// TwinCAT 3 PLC project TcoInspectors
// Title: TcoInspectors
// Company: Vortex.Library
// ProjectVersion: 0.6.0.913
// ProgramVersion: 3.1.4023.0
// libraries:
//   Tc2_Standard, * (Beckhoff Automation GmbH)
//   Tc2_System, * (Beckhoff Automation GmbH)
//   Tc2_Utilities, * (Beckhoff Automation GmbH)
//   Tc3_Module, * (Beckhoff Automation GmbH)
//   TcoCore, 0.6.0.913 (Vortex.Library)
// project tree:
//   / PlcTask.TcTTO
//   POUs/TcoInspector/ eTcoInspectorFailMode.TcDUT, IInspector.TcIO, IOnFail.TcIO, TcoComprehensiveResult.TcDUT, TcoInspector.TcPOU, TcoInspectorDialog.TcPOU, TcoInspectorTask.TcPOU, TcoInspectorData.TcDUT
//   POUs/TcoAnalogueInspector/ ITcoAnalogueInspector.TcIO, TcoAnalogueInspectorData.TcDUT, TcoAnalogueInspector.TcPOU
//   POUs/TcoDataInspector/ ITcoDataInspector.TcIO, TcoDataInspectorData.TcDUT, TcoDataInspector.TcPOU
//   POUs/ eOverallResult.TcDUT, eInspectorResult.TcDUT, MAIN.TcPOU
//   POUs/TcoDigitalInspector/ ITcoDigitalInspector.TcIO, TcoDigitalInspector.TcPOU, TcoDigitalInspectorData.TcDUT
//   POUs/TcoInspectionGroup/ ITcoInspectionGroup.TcIO, ITcoInspectionGroupAct.TcIO, TcoInspectionGroup.TcPOU
// real-time tasks:
//   TASK PlcTask: cycle T#10ms, priority 20, ADS port 350
//   TASK PlcTask1: cycle T#10ms, priority 21, ADS port 351

CONFIGURATION TcoInspectors
    RESOURCE PLC ON TwinCAT3
        TASK PlcTask(INTERVAL := T#10ms, PRIORITY := 20);
        PROGRAM MAIN WITH PlcTask : MAIN;
    END_RESOURCE
END_CONFIGURATION

// ---- POUs/TcoInspector/eTcoInspectorFailMode.TcDUT
{attribute 'qualified_only'}
{attribute 'strict'}
TYPE
    eTcoInspectorFailMode :
    (
        // On failed continues in the sequence but data are set to failed.
        CarryOn := 0,
        // Jump to specific step after first fail.
        JumpTo := 10,
        // Restores origin after first fail.
        Terminate := 20,
        // Retry when failed given number of times and continues in the sequence. Data are set to failed.
        RetryThenCarryOn := 30,
        // Retry, when failed given number of times abort sequence and continue in specifed step. Data are set to failed.
        RetryThenJumpTo := 40,
        // Retry, when failed given number of times abort sequence and continue with restore section. Data are set to failed.
        RetryThenTeminate := 50

    );
END_TYPE

// ---- POUs/TcoInspector/TcoComprehensiveResult.TcDUT
TYPE TcoComprehensiveResult :
STRUCT
    Result : eOverallResult;
    Failures : STRING(255);
    ErrorCodes : STRING(255);
END_STRUCT
END_TYPE

// ---- POUs/TcoInspector/TcoInspectorData.TcDUT
(*~
    <docu>
        <summary>
            Defines data commonly used accross different types of inspectors.
        </summary>
    </docu>
~*)
{attribute 'qlik_entity:Checks'}
{attribute 'qlik_ref_value_field:CheckName = AttributeHumanReadable'}
{attribute 'qlik_ref_value_field:StationName = AttributeQlikGroup'}
TYPE TcoInspectorData :
STRUCT
    (*~
        <docu>
        <summary>
            Inspection timestamp.
        </summary>
        </docu>
    ~*)
    {attribute addProperty Name "<#Time stamp#>"}
    {attribute clr [RenderIgnore("Control", "ShadowControl")]}
    {attribute 'qlik_load:TimeStamp'}
    TimeStamp : DT;
    (*~
        <docu>
        <summary>
            Pass time, elapses when the measured value has required value (see `ReuiredStatus`).
            The signal must have required value continuosly for this time span for the check to pass.
        </summary>
        </docu>
    ~*)
    {attribute addProperty Name "<#Stab.Time#>"}
    {attribute addProperty ToolTip "<#Stabilisation time. The inspection will pass when the condition is met continuously for the duration of this timespan.#>"}
    {attribute 'qlik_load:PassedTime'}
    PassTime : TIME;
    (*~
        <docu>
        <summary>
            Fail time. Is the maximum test duration (or timeout). If the condition for the successul test is not met within this time, the test fails.
        </summary>
        </docu>
    ~*)
    {attribute addProperty Name "<#Timeout#>"}
    {attribute addProperty ToolTip "<#Timeout. Maximal duration of the inspection within which the condition must be met.#>"}
    {attribute 'qlik_load:FailedTime'}
    FailTime : TIME;
    (*~
        <docu>
        <summary>
            Test result.
        </summary>
        </docu>
    ~*)
    {attribute addProperty Name "<#Result#>"}
    {attribute clr [RenderIgnore("Control", "ShadowControl")]}
    {attribute addProperty ToolTip "<#Result of the inspection.#>"}
    {attribute 'qlik_load:Result'}
    Result : eInspectorResult;
    (*~
        <docu>
        <summary>
            Test is excluded from evaluation. If TRUE the check is excluded, the test will run and provide detected value.
            Evaluation of excluded test should be handled by user code.
        </summary>
        </docu>
    ~*)
    {attribute addProperty Name "<#Exclude#>"}
    {attribute addProperty ToolTip "<#Inspection is excluded from the evaluation. The test will however run and provide detected value.#>"}
    {attribute 'qlik_load:IsExcluded'}
    IsExcluded : BOOL;
    (*~
        <docu>
        <summary>
            Test is bypassed, no eveluation occurs.
            Evaluation of excluded test should be handled by user code.
        </summary>
        </docu>
    ~*)
    {attribute addProperty Name "<#Bypass#>"}
    {attribute addProperty ToolTip "<#Test is bypassed, no eveluation occurs.#>"}
    {attribute 'qlik_load:IsByPassed'}
    IsByPassed : BOOL;
    (*~
        <docu>
        <summary>
            Verbatim description of the failure.
        </summary>
        </docu>
    ~*)
    {attribute addProperty Name "<#Failure description#>"}
    {attribute addProperty ToolTip "<#Brief failure desciption#>"}
    {attribute 'qlik_ignore'}
    FailureDescription : STRING(100);
    (*~
        <docu>
        <summary>
            Counter of allowed inspections.
        </summary>
        </docu>
    ~*)
    {attribute addProperty Name "<#Re-tries#>"}
    {attribute addProperty ToolTip "<#Inspection will repeat given number of times when inspection fails.#>"}
    {attribute 'qlik_load:NumberOfAllowedRetries'}
    NumberOfAllowedRetries : UINT;
    (*~
        <docu>
        <summary>
            Counter inspections.
        </summary>
        </docu>
    ~*)
    {attribute addProperty Name "<#Attempts#>"}
    {attribute addProperty ToolTip "<#Re-tries counter, count the number of times the inspection run on this inspector instance.#>"}
    {attribute 'qlik_load:RetryAttemptsCount'}
    RetryAttemptsCount : UINT;
    (*~
        <docu>
        <summary>
            Error code.
        </summary>
        </docu>
    ~*)
    {attribute addProperty Name "<#Code#>"}
    {attribute addProperty ToolTip "<#Arbitrary error code for this inspection#>"}
    {attribute 'qlik_load:ErrorCode'}
    ErrorCode : STRING(20);
END_STRUCT
END_TYPE

// ---- POUs/TcoDataInspector/TcoDataInspectorData.TcDUT
{attribute addProperty Name "AnalogueCheckerData"}
{attribute 'qlik_entity:Checks'}
{attribute 'qlik_ref_value_field:CheckName = AttributeHumanReadable'}
{attribute 'qlik_ref_value_field:StationName = AttributeQlikGroup'}
{attribute 'qlik_value_field:CheckType = Analogue'}
TYPE TcoDataInspectorData EXTENDS TcoInspectorData :
STRUCT
    (*~
        <docu>
        <summary>
            Required status for the check to Pass.
        </summary>
        </docu>
        ~*)
    {attribute addProperty Name "<#Required#>"}
    {attribute addProperty ToolTip "<#Required status for inspection to pass. Can contain pattern string when `Star notation is enabled`#>"}
    {attribute 'qlik_load:RequiredStatus'}
    RequiredStatus : STRING(255);
    (*~
        <docu>
        <summary>
            Detected status.
        </summary>
        </docu>
        ~*)
    {attribute addProperty  Name "<#Detected#>"}
    {attribute addProperty ToolTip "<#Detected data#>"}
    {attribute clr [RenderIgnore("Control", "ShadowControl", "ControlSlim", "ShadowControlSlim")]}
    {attribute 'qlik_load:Measured'}
    DetectedStatus : STRING(255);
    (*~
        <docu>
        <summary>
            When enabled (`true`) the date are evaluating with simple pattern matching.
        </summary>
        </docu>
        ~*)
    {attribute addProperty  Name "<*>"}
    {attribute addProperty ToolTip "<#Required status for inspection to pass. Can contain pattern string when `Star notation is enabled`#>"}
    {attribute 'qlik_load:Measured'}
    StarNotationEnabled : BOOL;
END_STRUCT
END_TYPE

// ---- POUs/eOverallResult.TcDUT
{attribute 'qualified_only'}
{attribute 'strict'}
TYPE eOverallResult :
(
    NoAction := 0,
    InProgress := 10,
    Passed := 20,
    Failed := 30
);
END_TYPE

// ---- POUs/TcoAnalogueInspector/TcoAnalogueInspectorData.TcDUT
{attribute addProperty Name "AnalogueCheckerData"}
{attribute addProperty Units ""}
{attribute 'qlik_entity:Checks'}
{attribute 'qlik_ref_value_field:CheckName = AttributeHumanReadable'}
{attribute 'qlik_ref_value_field:StationName = AttributeQlikGroup'}
{attribute 'qlik_value_field:CheckType = Analogue'}
TYPE TcoAnalogueInspectorData EXTENDS TcoInspectorData :
STRUCT
    (*~
        <docu>
        <summary>
            Required minimum value for the inspection to pass.
        </summary>
        </docu>
        ~*)
    {attribute addProperty  Name "<#Min.#>"}
    {attribute 'qlik_load:Minimum'}
    {attribute addProperty ToolTip "<#Min. value for the inspection to pass.#>"}
    RequiredMin : LREAL;
    (*~
        <docu>
        <summary>
            Detected status.
        </summary>
        </docu>
        ~*)
    {attribute addProperty  Name "<#Detected#>"}
    {attribute clr [RenderIgnore("Control", "ShadowControl", "ControlSlim", "ShadowControlSlim")]}
    {attribute addProperty ToolTip "<#Detected value#>"}
    {attribute 'qlik_load:Measured'}
    DetectedStatus : LREAL;
    (*~
        <docu>
        <summary>
            Required maximum value for the inspection to pass.
        </summary>
        </docu>
        ~*)
    {attribute addProperty  Name "<#Max.#>"}
    {attribute 'qlik_load:Maximum'}
    {attribute addProperty ToolTip "<#Max. value for the inspection to pass.#>"}
    RequiredMax : LREAL;
END_STRUCT
END_TYPE

// ---- POUs/TcoDigitalInspector/TcoDigitalInspectorData.TcDUT
{attribute addProperty Name "LogicCheckerData"}
{attribute 'qlik_value_field:CheckType = Logic'}
TYPE TcoDigitalInspectorData EXTENDS TcoInspectorData :
STRUCT
    (*~
        <docu>
        <summary>
            Required status for the check to Pass.
        </summary>
        </docu>
        ~*)
    {attribute addProperty Name "<#Required#>"}
    {attribute addProperty ToolTip "<#Sets the required status for the inspection to pass.#>"}
    {attribute 'qlik_load:RequiredStatus'}
    RequiredStatus : BOOL;
    (*~
        <docu>
        <summary>
            Detected status.
        </summary>
        </docu>
    ~*)
    {attribute addProperty Name "<#Detected#>"}
    {attribute clr [RenderIgnore("Control", "ShadowControl", "ControlSlim", "ShadowControlSlim")]}
    {attribute addProperty ToolTip "<#Displays detected status of this check.#>"}
    {attribute 'qlik_load:DetectedStatus'}
    DetectedStatus : BOOL;
END_STRUCT
END_TYPE

// ---- POUs/eInspectorResult.TcDUT
{attribute 'qualified_only'}
{attribute 'strict'}
TYPE eInspectorResult :
(
    NoAction := 0,
    Running := 10,
    Passed := 20,
    Failed := 30,
    Inconclusive := 35,
    Excluded := 40,
    Bypassed := 50
);
END_TYPE

// ---- POUs/TcoInspector/IInspector.TcIO
INTERFACE IInspector EXTENDS __SYSTEM.IQueryInterface

PROPERTY Busy : BOOL
GET
END_GET
END_PROPERTY

(*~
	<docu>
		<summary>
			Gets common data settings of inspectors.
		</summary>			
	</docu>	
~*)
PROPERTY CommonData : REFERENCE TO TcoInspectorData
GET
END_GET
END_PROPERTY

PROPERTY Coordinator : TcoCore.ITcoCoordinator
GET
END_GET
END_PROPERTY

PROPERTY Done : BOOL
GET
END_GET
END_PROPERTY

METHOD HideOverride : IInspector
END_METHOD

METHOD HideRetry : IInspector
END_METHOD

METHOD HideTerminate : IInspector
END_METHOD

PROPERTY Identity : ULINT
GET
END_GET
END_PROPERTY

METHOD Instruct : IInspector
VAR_INPUT
	inInstruction:STRING(255);
END_VAR
END_METHOD

METHOD InstructWithImage : IInspector
VAR_INPUT
	inImageSource:STRING(255);
	inHeight:REAL;
	inWidth:REAL;
END_VAR
END_METHOD

METHOD OnFail : IOnFail
END_METHOD

PROPERTY OverInspected : BOOL
GET
END_GET
END_PROPERTY

PROPERTY Result : eInspectorResult
GET
END_GET
END_PROPERTY

(*~
	<docu>
		<summary>
			Updates comprehensive result. The comprehensive result is set to `Failed` when any inspection fails or is inconclusive.
			Any bypassed or excluded inspection are not taken in the account.			
		</summary>			
	</docu>	
~*)
METHOD UpdateComprehensiveResult : IInspector
VAR_IN_OUT
	(*~
	<docu>
		<summary>
			Comprehensive result data structure to be updated.	
		</summary>			
	</docu>	
	~*)
    inoResult : TcoComprehensiveResult;
END_VAR
END_METHOD

(*~
	<docu>
		<summary>
			Provide information about the Inspector name (if there are multiple inspectors, only the failed ones will be displayed).  (e.g. {attribute addProperty Name "Bolt presence inspection"})
		</summary>			
	</docu>	
~*)
METHOD WithDescription : IInspector
END_METHOD

(*~
	<docu>
		<summary>
			Provide information about ErrorCode (if there are multiple inspectors, only the failed ones will be displayed). Error codes shoud be defined in Inspectors
		</summary>			
	</docu>	
~*)
METHOD WithErrorCode : IInspector
END_METHOD

(*~
	<docu>
		<summary>
			Provide information about Failure Description (if there are multiple inspectors, only the failed ones will be displayed). Failure description shoud be defined in Inspectors.
		</summary>			
	</docu>	
~*)
METHOD WithFailureDescription : IInspector
END_METHOD

END_INTERFACE

// ---- POUs/TcoInspector/IOnFail.TcIO
INTERFACE IOnFail EXTENDS __SYSTEM.IQueryInterface

METHOD CarryOn : BOOL
END_METHOD

METHOD Dialog : BOOL
VAR_INPUT
	inRetryStep : INT;
END_VAR
END_METHOD

METHOD DialogWithExternalClose : BOOL
VAR_INPUT
	inRetryStep : INT;
	inRetrySignal:BOOL;
	inTerminateSignal : BOOL;
END_VAR
END_METHOD

METHOD Evaluate : BOOL
VAR_INPUT
	inFromState : INT;
	inFailMode : eTcoInspectorFailMode;
    inToState : INT;
END_VAR
END_METHOD

METHOD Retry : BOOL
VAR_INPUT
	inFromState : INT;
END_VAR
END_METHOD

METHOD RetryThenTerminate : BOOL
VAR_INPUT
	inFromState : INT;
END_VAR
END_METHOD

METHOD Terminate : BOOL
END_METHOD

END_INTERFACE

// ---- POUs/TcoAnalogueInspector/ITcoAnalogueInspector.TcIO
INTERFACE ITcoAnalogueInspector

(*~
<docu>
<summary>
	Inspects the signal and evaluates that it matches the value set in `RequiredStatus`.
</summary>
<returns>
	Returns the interface with information about the state of inspection.
</returns>
</docu>
~*)
METHOD Inspect : IInspector
VAR_INPUT
    Status : LREAL;
END_VAR
END_METHOD

END_INTERFACE

// ---- POUs/TcoDataInspector/ITcoDataInspector.TcIO
INTERFACE ITcoDataInspector

(*~
<docu>
<summary>
	Inspects the signal and evaluates that it matches the value set in `RequiredStatus`.
</summary>
<returns>
	Returns the interface with information about the state of inspection.
</returns>
</docu>
~*)
METHOD Inspect : IInspector
VAR_INPUT
    Status : STRING(255);
END_VAR
END_METHOD

END_INTERFACE

// ---- POUs/TcoDigitalInspector/ITcoDigitalInspector.TcIO
INTERFACE ITcoDigitalInspector

(*~
<docu>
<summary>
	Inspects the signal and evaluates that it matches the value set in `RequiredStatus`.
</summary>
<returns>
	Returns the interface with information about the state of inspection.
</returns>
</docu>
~*)
METHOD Inspect : IInspector
VAR_INPUT
    Status : BOOL;
END_VAR
END_METHOD

END_INTERFACE

// ---- POUs/TcoInspectionGroup/ITcoInspectionGroup.TcIO
INTERFACE ITcoInspectionGroup

PROPERTY Done : BOOL
GET
END_GET
END_PROPERTY

METHOD Inspect : ITcoInspectionGroup
VAR_INPUT
    Inspector : IInspector;
END_VAR
END_METHOD

METHOD NormalizeRetries : ITcoInspectionGroup
VAR_INPUT
	inoInspection : IInspector;
END_VAR
END_METHOD

METHOD OnFail : IOnFail
END_METHOD

(*~
	<docu>
		<summary>
			Updates comprehensive result. The comprehensive result is set to `Failed` when any inspection fails or is inconclusive.
			Any bypassed or excluded inspection are not taken in the account.
		</summary>
	</docu>
~*)
METHOD UpdateComprehensiveResult : IInspector
VAR_IN_OUT
	(*~
	<docu>
		<summary>
			Comprehensive result data structure to be updated.
		</summary>
	</docu>
	~*)
    inoResult : TcoComprehensiveResult;
END_VAR
END_METHOD

END_INTERFACE

// ---- POUs/TcoInspectionGroup/ITcoInspectionGroupAct.TcIO
INTERFACE ITcoInspectionGroupAct

(*~
	<summary>
		Initiates grouped inspection.
	</summary>
~*)
METHOD Act : ITcoInspectionGroup
//VAR_IN_OUT
//	inoResult : TcoComprehensiveResult;
//END_VAR
END_METHOD

END_INTERFACE

// ---- POUs/MAIN.TcPOU
PROGRAM INTERNAL MAIN

END_PROGRAM

// ---- POUs/TcoInspector/TcoInspector.TcPOU
(*~
	<docu>
		<summary>
			Base block for signal and data inspectors. This block is abstract and must be inherited in derived block.
			Inspector provide a mechanism for detection and evaluation of various signals. The inspection is settable by a series of 
			settings, like stabilisation times, timeouts, repeats counts, etc.
		</summary>	
	</docu>	
~*)
FUNCTION_BLOCK ABSTRACT TcoInspector EXTENDS TcoCore.TcoObject IMPLEMENTS IInspector, IOnFail
VAR
	{attribute clr [CompilerOmits("BuilderPlainer", "BuilderShadowerInterface")]}
	_tcoInspectorDialogue : TcoInspectorDialog(THIS^);
	{attribute clr [CompilerOmits("BuilderPlainer", "BuilderShadowerInterface")]}
	_inspectorTask : TcoInspectorTask(THIS^);
	{attribute clr [CompilerOmits("BuilderPlainer", "BuilderShadowerInterface")]}	
	_coordinator    : TcoCore.ITcoCoordinator;
	{attribute 'hide'}	
	_isOverInspected : BOOL;
	{attribute 'hide'}	
	_tierUpdateOverall : TcoCore.TcoTier(THIS^);	
	{attribute 'hide'}	
	_originalOverallResult : TcoComprehensiveResult;
	{attribute 'hide'}	
	_refOverallResult : REFERENCE TO TcoComprehensiveResult;
END_VAR

METHOD PROTECTED _WithCoordinator : IInspector
VAR_INPUT
	inCoordinator : TcoCore.ITcoCoordinator;
END_VAR
_coordinator := inCoordinator;

IF(_coordinator.IsFreshState) THEN
	_inspectorTask.Restore();
	_tcoInspectorDialogue.Restore();
END_IF

_WithCoordinator := THIS^;
END_METHOD

(*~
	<docu>
		<summary>
			Gets `true` while the inspection is running.
		</summary>			
	</docu>	
~*)
PROPERTY PUBLIC Busy : BOOL
GET
Busy := _inspectorTask.Busy;
END_GET
END_PROPERTY

(*~
	<docu>
		<summary>
			Upon failure continues in the execution of coordinator. 
			The overall results is marked as failed.
		</summary>			
	</docu>	
~*)
{attribute 'hide'}
{attribute 'obsolete' := 'You should access `CarryOn` method via `OnFail()` method.'}
METHOD PUBLIC CarryOn : BOOL
IF(_coordinator = 0) THEN
	RETURN;			
END_IF

IF(THIS^.Done) THEN
	_coordinator.MoveNext();
END_IF;	
	
CarryOn := THIS^.Done;
END_METHOD

(*~
	<docu>
		<summary>
			Gets common data settings of inspectors.
		</summary>			
	</docu>	
~*)
PROPERTY ABSTRACT CommonData : REFERENCE TO TcoInspectorData
GET
END_GET
END_PROPERTY

(*~
	<docu>
		<summary>
			Gets the coordinator assotiated with this inspector. 
		</summary>			
	</docu>	
~*)
PROPERTY PUBLIC Coordinator : TcoCore.ITcoCoordinator
GET
Coordinator := _coordinator;
END_GET
END_PROPERTY

(*~
	<docu>
		<summary>
			Upon failure displays dialogue for the user to take decision about the fate of the inspection.			
		</summary>			
	</docu>	
~*)
METHOD PUBLIC Dialog : BOOL
VAR_INPUT
	inRetryStep : INT;
END_VAR
_tcoInspectorDialogue.Show(inRetryStep);
END_METHOD

(*~
	<docu>
		<summary>
			Upon failure displays dialogue for the user to take decision about the fate of the inspection.			
		</summary>			
	</docu>	
~*)
METHOD PUBLIC DialogWithExternalClose : BOOL
VAR_INPUT
	inRetryStep : INT;
	inRetrySignal:BOOL;
	inTerminateSignal : BOOL;
END_VAR
_tcoInspectorDialogue.ShowWithExternalClose(inRetryStep,inRetrySignal,inTerminateSignal);
END_METHOD

(*~
	<docu>
		<summary>
			Gets `true` when the inspection is done.
		</summary>			
	</docu>	
~*)
PROPERTY PUBLIC Done : BOOL
GET
Done := _inspectorTask.Done;
END_GET
END_PROPERTY

(*~
	<docu>
		<summary>
			Upon failure the inspection retries given number of time. When it reach	given numbers then terminate 		
		</summary>			
	</docu>	
~*)

{attribute 'hide'}
{attribute 'obsolete' := 'You should access `Evaluate` method via `OnFail()` method.'}
METHOD PUBLIC Evaluate : BOOL
VAR_INPUT
    (*~
	<docu>
		<summary>
			State from which the inspection will restart.		
		</summary>			
	</docu>	
	~*)
    inFromState : INT;
    (*~
	<docu>
		<summary>
			Behavior when ispection is failed		
		</summary>			
	</docu>	
	~*)
    inFailMode : eTcoInspectorFailMode;
    (*~
	<docu>
		<summary>
			State from which the inspection will continue.		
		</summary>			
	</docu>	
	~*)
    inToState : INT;
END_VAR
IF (_coordinator = 0) THEN
    RETURN;
END_IF

IF (THIS^.Done) THEN
    IF (THIS^.Result = eInspectorResult.Failed) THEN
        IF (__ISVALIDREF(_refOverallResult)) THEN
            _refOverallResult := _originalOverallResult;
        END_IF

        IF inFailMode = eTcoInspectorFailMode.CarryOn THEN
            _coordinator.MoveNext();
        ELSIF inFailMode = eTcoInspectorFailMode.JumpTo THEN
            _coordinator.Retry(inToState);
        ELSIF inFailMode = eTcoInspectorFailMode.Terminate THEN
            _coordinator.Terminate();
        ELSIF inFailMode = eTcoInspectorFailMode.RetryThenCarryOn THEN
            IF OverInspected THEN
                _coordinator.MoveNext();
            ELSE
                _coordinator.Retry(inFromState);
            END_IF;
        ELSIF inFailMode = eTcoInspectorFailMode.RetryThenJumpTo THEN
            IF OverInspected THEN
                _coordinator.Retry(inToState);
            ELSE
                _coordinator.Retry(inFromState);
            END_IF;

        ELSIF inFailMode = eTcoInspectorFailMode.RetryThenTeminate THEN
            IF OverInspected THEN
                _coordinator.Terminate();
            ELSE
                _coordinator.Retry(inFromState);
            END_IF;

        END_IF
    ELSE

        _coordinator.MoveNext();
    END_IF;
END_IF;

Evaluate := THIS^.Done;
END_METHOD

{attribute 'hide'}
METHOD PUBLIC FB_init : BOOL
VAR_INPUT
	bInitRetains : BOOL; // if TRUE, the retain variables are initialized (warm start / cold start)
	bInCopyCode : BOOL;  // if TRUE, the instance afterwards gets moved into the copy code (online change)
	ParentObject : ITcoObject;
END_VAR
//// Hate to do this guys but I get compile error, seems to be a bug in tc
//
END_METHOD

(*~
	<docu>
		<summary>
			Provide option to hide override button. Default state is  visible. 
		</summary>			
	</docu>	
~*)
METHOD HideOverride : IInspector

HideOverride := THIS^;

_tcoInspectorDialogue.HideTetminate:=TRUE;
END_METHOD

(*~
	<docu>
		<summary>
			Provide option to hide retry button. Default state is  visible. 
		</summary>			
	</docu>	
~*)
METHOD HideRetry : IInspector

HideRetry := THIS^;

_tcoInspectorDialogue.HideRetry:=TRUE;
END_METHOD

(*~
	<docu>
		<summary>
			Provide option to hide terminate button. Default state is  visible. 
		</summary>			
	</docu>	
~*)
METHOD HideTerminate : IInspector

HideTerminate := THIS^;

_tcoInspectorDialogue.HideTetminate:=TRUE;
END_METHOD

METHOD PUBLIC Instruct:IInspector
VAR_INPUT
	inInstruction:STRING(255);
END_VAR

Instruct := THIS^;

_tcoInspectorDialogue.SetInstruction(inInstruction);
END_METHOD

METHOD PUBLIC InstructWithImage:IInspector
VAR_INPUT
	inImageSource:STRING(255);
	inHeight:REAL;
	inWidth:REAL;
END_VAR

InstructWithImage := THIS^;

_tcoInspectorDialogue.SetImageSource(inImageSource,inHeight,inWidth);
END_METHOD

(*~
	<docu>
		<summary>
			Gets `true` when this inspection overruns max number of inspection.
		</summary>			
	</docu>	
~*)
METHOD PROTECTED IsOverinspected : BOOL
_isOverInspected := THIS^.OverInspected;
IF(OverInspected) THEN			
	THIS^._inspectorTask.Invoke();
	IF(THIS^._inspectorTask.Execute()) THEN		
		THIS^._inspectorTask.InspectionData.Result := eInspectorResult.Failed;
		THIS^._inspectorTask.DoneWhen(TRUE);	
	END_IF	
END_IF

IsOverinspected := OverInspected;
END_METHOD

(*~
	<docu>
		<summary>
			Executes each time the `Inspect` method is called.
		</summary>			
	</docu>	
~*)
METHOD PROTECTED FINAL OnEnterInspection : BOOL
VAR_INPUT
END_VAR
THIS^._tcoInspectorDialogue.SetInspector(THIS^);
END_METHOD

METHOD PUBLIC OnFail : IOnFail
IF(_coordinator = 0) THEN
	Messenger.Programming('Missing `coordinator`. You will need to call inspector `WithCoordinator` method.');			
END_IF

OnFail := THIS^;
END_METHOD

(*~
	<docu>
		<summary>
			Gets `true` when the number of inspections excceds `NumberOfAllowedRetries`.
		</summary>			
	</docu>	
~*)
PROPERTY PUBLIC OverInspected : BOOL
GET
IF(__ISVALIDREF(_inspectorTask._inspectionData)) THEN
	OverInspected := (_inspectorTask._inspectionData.RetryAttemptsCount >= _inspectorTask._inspectionData.NumberOfAllowedRetries) 
					 AND (_inspectorTask._inspectionData.NumberOfAllowedRetries <> 0);
END_IF;
END_GET
END_PROPERTY

METHOD Restore : TcoCore.ITcoRestorable
VAR_INPUT
END_VAR
_tcoInspectorDialogue.Restore();
END_METHOD

(*~
	<docu>
		<summary>
			Gets the inspection result of this inspector.
		</summary>			
	</docu>	
~*)
PROPERTY PUBLIC Result : eInspectorResult
GET
IF(__ISVALIDREF(_inspectorTask._inspectionData)) THEN
	Result := _inspectorTask._inspectionData.Result;	
END_IF;
END_GET
END_PROPERTY

(*~
	<docu>
		<summary>
			Upon failure the inspection retries given number of time.			
		</summary>			
	</docu>	
~*)
{attribute 'hide'}
{attribute 'obsolete' := 'You should access `Retry` method via `OnFail()` method.'}
METHOD PUBLIC Retry : BOOL
VAR_INPUT
	(*~
	<docu>
		<summary>
			State from which the inspection will restart.		
		</summary>			
	</docu>	
	~*)
	inFromState : INT;
END_VAR
IF(_coordinator = 0) THEN
	RETURN;	
END_IF

IF(THIS^.Done) THEN
	IF(THIS^.Result = eInspectorResult.Failed) THEN
		IF(__ISVALIDREF(_refOverallResult)) THEN
			_refOverallResult := _originalOverallResult;
		END_IF
		_coordinator.Retry(inFromState);
	ELSE
		_coordinator.MoveNext();
	END_IF;	
END_IF;	


Retry := THIS^.Done;
END_METHOD

(*~
	<docu>
		<summary>
			Upon failure the inspection retries given number of time. When it reach	given numbers then terminate 		
		</summary>			
	</docu>	
~*)

{attribute 'hide'}
{attribute 'obsolete' := 'You should access `Retry` method via `OnFail()` method.'}
METHOD PUBLIC RetryThenTerminate : BOOL
VAR_INPUT
	(*~
	<docu>
		<summary>
			State from which the inspection will restart.		
		</summary>			
	</docu>	
	~*)
	inFromState : INT;
END_VAR
IF(_coordinator = 0) THEN
	RETURN;	
END_IF

IF(THIS^.Done) THEN
	IF(THIS^.Result = eInspectorResult.Failed) THEN
		IF(__ISVALIDREF(_refOverallResult)) THEN
			_refOverallResult := _originalOverallResult;
		END_IF
		
		IF OverInspected THEN
			_coordinator.Terminate();
		ELSE
			_coordinator.Retry(inFromState);
		END_IF
	ELSE
		_coordinator.MoveNext();
	END_IF;	
END_IF;	


RetryThenTerminate := THIS^.Done;
END_METHOD

(*~
	<docu>
		<summary>
			Upon failure the inspection terminates the run of the coordinator.			
		</summary>			
	</docu>	
~*)
{attribute 'hide'}
{attribute 'obsolete' := 'You should access `Terminate` method via `OnFail()` method.'}
METHOD PUBLIC Terminate : BOOL
IF(_coordinator = 0) THEN
	RETURN;	
END_IF

IF(THIS^.Done) THEN
	IF(THIS^.Result = eInspectorResult.Failed) THEN
		_coordinator.Terminate();
	ELSE
		_coordinator.MoveNext();
	END_IF;	
END_IF;	

Terminate := THIS^.Done;
END_METHOD

(*~
	<docu>
		<summary>
			Updates comprehensive result. The comprehensive result is set to `Failed` when any inspection fails or is inconclusive.
			Any bypassed or excluded inspection are not taken in the account.			
		</summary>			
	</docu>	
~*)
{attribute 'hide'}
{attribute 'obsolete' := 'You should access `UpdateOverall` property via `Inspect` method.'}
METHOD PUBLIC UpdateComprehensiveResult : IInspector
VAR_IN_OUT
	(*~
	<docu>
		<summary>
			Comprehensive result data structure to be updated.	
		</summary>			
	</docu>	
	~*)
    inoResult : TcoComprehensiveResult;
END_VAR
UpdateComprehensiveResult := THIS^;

IF(_tierUpdateOverall.IsNewTier()) THEN	
	_refOverallResult REF= inoResult;
	_originalOverallResult := inoResult;
END_IF


IF (NOT __ISVALIDREF(_inspectorTask.InspectionData)) THEN
    inoResult.Result := eOverallResult.NoAction;
    RETURN;
END_IF

CASE _inspectorTask.InspectionData.Result OF
    eInspectorResult.NoAction:
        ;
    eInspectorResult.Running:
        ;
    eInspectorResult.Passed:
        ;
    eInspectorResult.Failed:
        inoResult.Result   := eOverallResult.Failed;
		UpdateDescriptions(inoResult);		       			
    eInspectorResult.Inconclusive:
        inoResult.Result := eOverallResult.Failed;
		UpdateDescriptions(inoResult);
    eInspectorResult.Excluded:
        ;
    eInspectorResult.Bypassed:
        ;
END_CASE
END_METHOD

(*~
	<docu>
		<summary>
			Updates failure description. Adding `FailureDescription` do the overall result structure.
		</summary>	
	</docu>	
~*)
METHOD PROTECTED UpdateDescriptions
VAR_IN_OUT
	inoResult : TcoComprehensiveResult;
END_VAR
IF(_inspectorTask.OnDoneFlag) THEN
	inoResult.Failures := THIS^.Context.Environment.Messaging.StringBuilder.Clear()
				.Append(inoResult.Failures)				
				.Append(_inspectorTask.InspectionData.FailureDescription)
				.Append(';')
				.ToString();
	
	inoResult.ErrorCodes := THIS^.Context.Environment.Messaging.StringBuilder.Clear()
				.Append(inoResult.ErrorCodes)				
				.Append(_inspectorTask.InspectionData.ErrorCode)
				.Append(';')
				.ToString();	
END_IF;
END_METHOD

(*~
	<docu>
		<summary>
			Provide information(name defined in attribute name) about failed inspection (if there are multiple inspectors, only the failed ones will be displayed). 
		</summary>			
	</docu>	
~*)
METHOD WithDescription : IInspector

WithDescription := THIS^;

_tcoInspectorDialogue.ShowDescription:=TRUE;
END_METHOD

(*~
	<docu>
		<summary>
			Provide information about ErrorCode (if there are multiple inspectors, only the failed ones will be displayed). Error codes shoud be defined in Inspectors
		</summary>			
	</docu>	
~*)
METHOD WithErrorCode : IInspector

WithErrorCode := THIS^;

_tcoInspectorDialogue.ShowErrorCode:=TRUE;
END_METHOD

(*~
	<docu>
		<summary>
			Provide information about Failure Description (if there are multiple inspectors, only the failed ones will be displayed). Failure description shoud be defined in Inspectors.
		</summary>			
	</docu>	
~*)
METHOD WithFailureDescription : IInspector

WithFailureDescription := THIS^;

_tcoInspectorDialogue.ShowFailureDescription:=TRUE;
END_METHOD

END_FUNCTION_BLOCK

// ---- POUs/TcoInspector/TcoInspectorDialog.TcPOU
(*~
	<docu>
		<summary>
			Provides dialog with the user to allow for deciding how to proceed in case of failure.	
		</summary>	
	</docu>	
~*)
FUNCTION_BLOCK PUBLIC TcoInspectorDialog EXTENDS TcoCore.TcoDialogBase
VAR
    _dialogRetry : BOOL;
    _dialogTerminate : BOOL;
    _dialogOverride : BOOL;
    _dialogIsClosed : BOOL;
    _isOverInspected : BOOL;
    {attribute 'hide'}
    _refInspector : REFERENCE TO TcoInspector;
    {attribute 'hide'}
    _tierAct : TcoCore.TcoTier(THIS^);

    _rTrigRetry : R_TRIG;
    _rTrigTerminate : R_TRIG;
    _externalCloseReq : BOOL;
    _closeRetrySignal : BOOL;
    _closeTerminateSignal : BOOL;

    _instruction : STRING(255);
    _source : STRING(255);
    _imageHeight : REAL;
    _imageWidth : REAL;
    _hideOverideButton : BOOL;
    _hideTerminateButton : BOOL;
    _hideRetryButton : BOOL;

    _showFailureDescription : BOOL;
    _showErrorCode : BOOL;
    _showDescription : BOOL;

    _isInvoked : BOOL;
END_VAR

SUPER^();

PROPERTY DialogIsClosed: REFERENCE TO BOOL
GET
DialogIsClosed ref=_dialogIsClosed;
END_GET
END_PROPERTY

PROPERTY DialogOverride: REFERENCE TO BOOL
GET
DialogOverride ref=_dialogOverride;
END_GET
END_PROPERTY

PROPERTY DialogRetry: REFERENCE TO BOOL
GET
DialogRetry ref=_dialogRetry;
END_GET
END_PROPERTY

PROPERTY DialogTerminate: REFERENCE TO BOOL
GET
DialogTerminate ref=_dialogTerminate;
END_GET
END_PROPERTY

{attribute 'hide'}
METHOD PUBLIC FB_init : BOOL
VAR_INPUT
	bInitRetains : BOOL; // if TRUE, the retain variables are initialized (warm start / cold start)
	bInCopyCode : BOOL;  // if TRUE, the instance afterwards gets moved into the copy code (online change)
	ParentObject : ITcoObject;
END_VAR
END_METHOD

METHOD HandleExternalSignals
VAR_INPUT
	inRetrySignal:BOOL;
	inTerminateSignal : BOOL;
	
END_VAR

_closeRetrySignal:=FALSE;
_closeTerminateSignal:=FALSE;


_rTrigRetry(CLK:=inRetrySignal);
IF _rTrigRetry.q THEN
	_closeRetrySignal:=TRUE;
END_IF

_rTrigTerminate(CLK:=inTerminateSignal);
IF _rTrigTerminate.q THEN
	_closeTerminateSignal:=TRUE;
END_IF

 IF(_refInspector.Done) THEN	
	 	IF NOT ( _dialogRetry) THEN
			_dialogRetry:=_closeRetrySignal;
		END_IF;
		IF NOT ( _dialogTerminate) THEN
			_dialogTerminate:=_closeTerminateSignal;
		END_IF;
 END_IF
END_METHOD

PROPERTY HideOverride: REFERENCE TO BOOL
GET
HideOverride ref=_hideOverideButton;
END_GET
END_PROPERTY

PROPERTY HideRetry: REFERENCE TO BOOL
GET
HideRetry ref=_hideRetryButton;
END_GET
END_PROPERTY

PROPERTY HideTetminate: REFERENCE TO BOOL
GET
HideTetminate ref=_hideTerminateButton;
END_GET
END_PROPERTY

METHOD PROTECTED OnStart
SUPER^.OnStart();
_isInvoked:=TRUE;
_dialogIsClosed:=FALSE;
_dialogRetry	    :=  FALSE;	
_dialogTerminate  	:=  FALSE;	
_dialogOverride   	:=  FALSE;
END_METHOD

PROPERTY INTERNAL OverInspected : BOOL
GET
OverInspected := _isOverInspected;
END_GET
SET
_isOverInspected := OverInspected;
END_SET
END_PROPERTY

METHOD Restore : TcoCore.ITcoRestorable
VAR_INPUT
END_VAR
SUPER^.Restore();
_dialogRetry	    :=  FALSE;	
_dialogTerminate  	:=  FALSE;	
_dialogOverride   	:=  FALSE;

_instruction:='';
_source:='';
_hideOverideButton:=FALSE;
_hideRetryButton:=FALSE;
_hideTerminateButton:=FALSE;
_imageHeight:=400;
_imageWidth:=600;
_showDescription:=FALSE;
_showFailureDescription:=FALSE;
_showErrorCode:=FALSE;
_isInvoked:=FALSE;
END_METHOD

METHOD SetImageSource
VAR_INPUT
	inSource:STRING(255);
	inHeight:REAL;
	inWidth:REAL;
END_VAR
_source:=inSource;
_imageHeight:=inHeight;
_imageWidth:= inWidth;
END_METHOD

METHOD SetInspector
VAR_INPUT 
	refInspector : REFERENCE TO TcoInspector;
END_VAR
_refInspector REF= refInspector;
END_METHOD

METHOD SetInstruction
VAR_INPUT
	inInstruction:STRING(255);
END_VAR
_instruction:=inInstruction;
END_METHOD

METHOD Show
VAR_INPUT
	inRetryStep : INT;
END_VAR
_isOverInspected := _refInspector.OverInspected;

IF(_tierAct.IsNewTier()) THEN
	THIS^.Restore();
END_IF

 IF(_refInspector.Done) THEN		
	IF(_refInspector.Result = eInspectorResult.Failed) THEN
		THIS^.Invoke();
		SUPER^();	
		{warning disable C0357}
		IF(_dialogRetry AND _dialogIsClosed) THEN
			_isInvoked:=FALSE;
			_refInspector.Retry(inRetryStep);
		END_IF
		
		IF(_dialogTerminate AND _dialogIsClosed) THEN
			_isInvoked:=FALSE;
			_refInspector.Terminate();
		END_IF
		
		IF(_dialogOverride AND _dialogIsClosed) THEN
			_isInvoked:=FALSE;
			_refInspector.CarryOn();
		END_IF
		{warning enable C0357}
	ELSE
		IF(_refInspector.Coordinator <> 0) THEN
			_refInspector.Coordinator.MoveNext();
		END_IF;	
	END_IF;	
END_IF;

IF THIS^._taskState=eTaskState.Done 
		AND ( _dialogRetry
		OR _dialogTerminate
		OR _dialogOverride)
		and _dialogIsClosed  THEN	
	THIS^.Restore();
END_IF;
END_METHOD

PROPERTY ShowDescription: REFERENCE TO BOOL
GET
ShowDescription ref=_showDescription;
END_GET
END_PROPERTY

PROPERTY ShowErrorCode: REFERENCE TO BOOL
GET
ShowErrorCode ref=_showErrorCode;
END_GET
END_PROPERTY

PROPERTY ShowFailureDescription: REFERENCE TO BOOL
GET
ShowFailureDescription ref=_showFailureDescription;
END_GET
END_PROPERTY

METHOD ShowWithExternalClose
VAR_INPUT
	inRetryStep : INT;
	inRetrySignal:BOOL;
	inTerminateSignal : BOOL;
	
END_VAR
//IF THIS^._taskState=eTaskState.Ready THEN
//	_dialogRetry	    	:=  FALSE;	
//	_dialogTerminate  	:=  FALSE;	
//	_dialogOverride   	:=  FALSE;
//END_IF

_isOverInspected := _refInspector.OverInspected;

IF(_tierAct.IsNewTier()) THEN
	THIS^.Restore();
END_IF

HandleExternalSignals(inRetrySignal:=inRetrySignal,inTerminateSignal:=inTerminateSignal);


 IF(_refInspector.Done) THEN		
	IF(_refInspector.Result = eInspectorResult.Failed) THEN
		THIS^.Invoke();
		SUPER^();	
		{warning disable C0357}
		//retry
	
		
		IF(_dialogRetry AND _dialogIsClosed) THEN
			_isInvoked:=FALSE;
			_refInspector.Retry(inRetryStep);
		END_IF
		//terminate
		
		IF(_dialogTerminate  AND  _dialogIsClosed) THEN
			_isInvoked:=FALSE;
			_refInspector.Terminate();
		END_IF
		
		IF(_dialogOverride AND _dialogIsClosed) THEN
			_isInvoked:=FALSE;
			_refInspector.CarryOn();
		END_IF
		{warning enable C0357}
	ELSE
		IF(_refInspector.Coordinator <> 0) THEN
			_refInspector.Coordinator.MoveNext();
		END_IF;	
	END_IF;	
END_IF;


IF THIS^._taskState=eTaskState.Done 
		AND ( _dialogRetry
		OR _dialogTerminate
		OR _dialogOverride)
		and _dialogIsClosed  THEN	
	THIS^.Restore();
END_IF;
END_METHOD

END_FUNCTION_BLOCK

// ---- POUs/TcoInspector/TcoInspectorTask.TcPOU
(*~
    <docu>
        <summary>
            Base block for inspectors.
        </summary>
    </docu>
~*)
FUNCTION_BLOCK TcoInspectorTask EXTENDS TcoCore.TcoTask
VAR
    _inspectionData : REFERENCE TO TcoInspectorData;
    _passTimer : Tc2_Standard.TON;
    _failTimer : Tc2_Standard.TON;
    _onDoneFlag : BOOL;
END_VAR

(*~
    <docu>
        <summary>
            Returns true if the task is Busy, otherwise false.
            This method needs to be called cyclically.
        </summary>
    </docu>
~*)
METHOD Execute : BOOL
VAR
    _serviceableParent : ITcoServiceable;
END_VAR
VAR
    tmpTimeDiff : TIME;
END_VAR
_onDoneFlag := FALSE;
Execute := SUPER^.Execute();
END_METHOD

{attribute 'hide'}
METHOD PUBLIC FB_init : BOOL
VAR_INPUT
    bInitRetains : BOOL; // if TRUE, the retain variables are initialized (warm start / cold start)
    bInCopyCode : BOOL; // if TRUE, the instance afterwards gets moved into the copy code (online change)
    ParentObject : ITcoObject;
END_VAR
//// Hate to do this guys but I get compile error, seems to be a bug in tc
//
END_METHOD

PROPERTY InspectionData : REFERENCE TO TcoInspectorData
GET
InspectionData REF= _inspectionData;
END_GET
SET
_inspectionData REF= InspectionData;
END_SET
END_PROPERTY

(*~
    <docu>
        <summary>
            Executes when task reaches the ```Done``` state .
        </summary>
    </docu>
~*)
METHOD PROTECTED OnDone
SUPER^.OnDone();
_inspectionData.RetryAttemptsCount := _inspectionData.RetryAttemptsCount + 1;

IF (_inspectionData.Result = eInspectorResult.Bypassed) THEN
    RETURN;
END_IF;

_inspectionData.TimeStamp := Context.RealTimeClock.NowLocal();
_inspectionData.Result := eInspectorResult.Failed;

IF (NOT _failTimer.Q AND _passTimer.Q) THEN
    _inspectionData.Result := eInspectorResult.Passed;
END_IF

IF (_inspectionData.IsExcluded) THEN
    _inspectionData.Result := eInspectorResult.Excluded;
END_IF

_onDoneFlag := TRUE;
END_METHOD

PROPERTY OnDoneFlag : BOOL
GET
OnDoneFlag := _onDoneFlag;
END_GET
END_PROPERTY

(*~
    <docu>
        <summary>
            Executes once when inspection starts.
        </summary>
    </docu>
~*)
METHOD PROTECTED OnStart
SUPER^.OnStart();

IF (_inspectionData.PassTime = T#0S) THEN
    _inspectionData.PassTime := T#50MS;
END_IF;

IF (_inspectionData.FailTime = T#0S) THEN
    _inspectionData.FailTime := T#100MS;
END_IF;

_inspectionData.Result := eInspectorResult.NoAction;
_passTimer(IN := FALSE, PT := T#0MS);
_failTimer(IN := FALSE, PT := T#0MS);
END_METHOD

(*~
    <docu>
        <summary>
            Restores this instance to the Ready state. Can be called explicitly or from within one of the restore mechanisms.
            <para>
                See also <see cref="PlcDocu.TcoCore.TcoTask.AutoRestorable()"/>
            </para>
        </summary>
    </docu>
~*)
METHOD Restore : ITcoRestorable
SUPER^.Restore();
_onDoneFlag := FALSE;
END_METHOD

END_FUNCTION_BLOCK

// ---- POUs/TcoDataInspector/TcoDataInspector.TcPOU
(*~
<docu>
<summary>
	Provides a mechanism for inspecting status of discrete signal.	
</summary>
</docu>
~*)
FUNCTION_BLOCK TcoDataInspector EXTENDS TcoInspector IMPLEMENTS ITcoDataInspector
VAR
    _data : TcoDataInspectorData;
	{attribute 'hide'}
	_lastOutValue : STRING;
END_VAR

(*~
	<docu>
		<summary>
			Gets common data settings of inspectors.
		</summary>			
	</docu>	
~*)
PROPERTY CommonData : REFERENCE TO TcoInspectorData
GET
CommonData REF= _data;
END_GET
END_PROPERTY

(*~
<docu>
<summary>
	Gets data of this inspector.
</summary>
</docu>
~*)
PROPERTY Data : REFERENCE TO TcoDataInspectorData
GET
Data REF= _data;
END_GET
END_PROPERTY

(*~
<docu>
<summary>
	Inspects the signal and evaluates that it matches the value set in `RequiredStatus`.
</summary>
<returns>
	Returns the interface with information about the state of inspection.
</returns>
</docu>
~*)
METHOD Inspect : IInspector
VAR_INPUT
    Status : STRING(255);
END_VAR

VAR
	tmpResult : BOOL;
	charIndex : INT;
	charRequired : STRING(1);
	charAcquired : STRING(1);	
END_VAR

VAR CONSTANT
    epsilon : REAL := 1;
END_VAR
Inspect := THIS^;

_inspectorTask.InspectionData REF= _data;

OnEnterInspection();

IF(IsOverinspected())THEN
	RETURN;
END_IF


_inspectorTask.Invoke();

IF (_inspectorTask.Execute()) THEN
    IF (_data.IsByPassed) THEN
        _data.Result    := eInspectorResult.Bypassed;
        _data.TimeStamp := Context.RealTimeClock.NowLocal();
        _inspectorTask.DoneWhen(TRUE);
        RETURN;
    END_IF
		
	    _data.Result := eInspectorResult.Running;
	
		THIS^.Messenger.OnCondition(LEN(Status) > 250 OR LEN(_data.RequiredStatus) > 250).Build().Append('The checked input string or required pattern string exceeds 250 characters.').As().AsError();
		
        IF(LEN(Status) > 250 OR LEN(_data.RequiredStatus) > 254) THEN                
            RETURN;
        END_IF
		
	    _data.DetectedStatus := Status;
		
		
		IF(_data.StarNotationEnabled) THEN
			tmpResult := TRUE;
			FOR charIndex := 1 TO LEN(_data.RequiredStatus) DO
				charRequired := MID(_data.RequiredStatus, 1, charIndex);
				
				IF(LEN(_data.DetectedStatus) >= charIndex) THEN
					charAcquired :=  MID(_data.DetectedStatus, 1, charIndex);
				ELSE
					charAcquired := '';
				END_IF;	
				
				IF(charRequired <> '*' AND charRequired <> '#') THEN
					tmpResult := charRequired = charAcquired;
				ELSIF(charRequired = '#') THEN
					tmpResult := IsNumber(charAcquired);            	
				END_IF
				
				IF(NOT tmpResult) THEN
					EXIT;
				END_IF				
			END_FOR
		ELSE
			
			tmpResult := F_RTrim(_data.DetectedStatus) =F_RTrim(_data.RequiredStatus);	
		END_IF
		
       
		IF(NOT tmpResult) THEN	
			_lastOutValue := Status;
		END_IF
		
		_inspectorTask._failTimer(IN:= TRUE, PT:=_data.FailTime);
		_inspectorTask._passTimer(IN:= tmpResult,PT:=_data.PassTime);
									  
     	IF(_inspectorTask._failTimer.Q OR _inspectorTask._passTimer.Q) THEN	  
     		_inspectorTask.DoneWhen(TRUE);
			OnDone();
	 	END_IF;	
END_IF;
END_METHOD

METHOD PROTECTED IsNumber : BOOL
VAR_INPUT
    inCharacter : STRING(1);
END_VAR
VAR
    numericalRapresentation : BYTE;
END_VAR
IF (inCharacter = '0'
OR  inCharacter = '1'
OR  inCharacter = '2'
OR  inCharacter = '3'
OR  inCharacter = '4'
OR  inCharacter = '5'
OR  inCharacter = '6'
OR  inCharacter = '7'
OR  inCharacter = '8'
OR  inCharacter = '9') 
THEN
	IsNumber := TRUE;
	RETURN;
END_IF;

IsNumber := FALSE;
END_METHOD

(*~
	<docu>
		<summary>
			Executes when task reaches the ```Done``` state .
		</summary>			
	</docu>	
~*)
METHOD PROTECTED OnDone
IF (_data.Result = eInspectorResult.Failed) THEN
     _data.DetectedStatus := _lastOutValue;
END_IF
END_METHOD

METHOD WithCoordinator : ITcoDataInspector
VAR_INPUT
	inCoordinator : TcoCore.ITcoCoordinator;
END_VAR
_WithCoordinator(inCoordinator);
WithCoordinator := THIS^;
END_METHOD

END_FUNCTION_BLOCK

// ---- POUs/TcoAnalogueInspector/TcoAnalogueInspector.TcPOU
(*~
<docu>
<summary>
    Provides a mechanism for inspecting status of discrete signal.
</summary>
</docu>
~*)
FUNCTION_BLOCK TcoAnalogueInspector EXTENDS TcoInspector IMPLEMENTS ITcoAnalogueInspector
VAR
    _data : TcoAnalogueInspectorData;
    {attribute 'hide'}
    _lastOutValue : LREAL;
END_VAR

(*~
    <docu>
        <summary>
            Gets common data settings of inspectors.
        </summary>
    </docu>
~*)
PROPERTY CommonData : REFERENCE TO TcoInspectorData
GET
CommonData REF= _data;
END_GET
END_PROPERTY

(*~
<docu>
<summary>
    Gets data of this inspector.
</summary>
</docu>
~*)
PROPERTY Data : REFERENCE TO TcoAnalogueInspectorData
GET
Data REF= _data;
END_GET
END_PROPERTY

(*~
<docu>
<summary>
    Inspects the signal and evaluates that it matches the value set in `RequiredStatus`.
</summary>
<returns>
    Returns the interface with information about the state of inspection.
</returns>
</docu>
~*)
METHOD Inspect : IInspector
VAR_INPUT
    Status : LREAL;
END_VAR
VAR
    tmpResult : BOOL;
    _minimum : LREAL;
    _value : LREAL;
    _maximum : LREAL;
END_VAR
VAR CONSTANT
    epsilon : REAL := 100000;
END_VAR
Inspect := THIS^;
_inspectorTask.InspectionData REF= _data;
OnEnterInspection();

IF (IsOverinspected()) THEN
    RETURN;
END_IF

_inspectorTask.Invoke();

IF (_inspectorTask.Execute()) THEN
    IF (_data.IsByPassed) THEN
        _data.Result := eInspectorResult.Bypassed;
        _data.TimeStamp := Context.RealTimeClock.NowLocal();
        _inspectorTask.DoneWhen(TRUE);
        RETURN;
    END_IF

    _data.Result := eInspectorResult.Running;
    _minimum := (Data.RequiredMin * epsilon);
    _value := (Status * epsilon);
    _maximum := (Data.RequiredMax * epsilon);
    Data.DetectedStatus := Status;
    tmpResult := (_minimum <= _value) AND (_maximum >= _value);

    IF (NOT tmpResult) THEN
        _lastOutValue := Status;
    END_IF

    _inspectorTask._failTimer(IN := TRUE, PT := _data.FailTime);
    _inspectorTask._passTimer(IN := tmpResult, PT := _data.PassTime);

    IF (_inspectorTask._failTimer.Q OR _inspectorTask._passTimer.Q) THEN
        _inspectorTask.DoneWhen(TRUE);
        OnDone();
    END_IF;
END_IF;
END_METHOD

(*~
    <docu>
        <summary>
            Executes when task reaches the ```Done``` state .
        </summary>
    </docu>
~*)
METHOD PROTECTED OnDone
IF (_data.Result = eInspectorResult.Failed) THEN
    _data.DetectedStatus := _lastOutValue;
END_IF
END_METHOD

METHOD WithCoordinator : ITcoAnalogueInspector
VAR_INPUT
    inCoordinator : TcoCore.ITcoCoordinator;
END_VAR
_WithCoordinator(inCoordinator);
WithCoordinator := THIS^;
END_METHOD

END_FUNCTION_BLOCK

// ---- POUs/TcoDigitalInspector/TcoDigitalInspector.TcPOU
(*~
    <docu>
    <summary>
        Provides a mechanism for inspecting status of discrete signal.
    </summary>
    <example>
        [!code-pas[StandardDialog](~/../TcOpen/src/TcoInspectors/src/XAE/XAE/TcoInspectorsTests/POUs/Examples/ExampleContext.TcPOU?name=StandardDialog)]
        [!code-csharp[DialogInitialization](~/../TcOpen/src/TcoInspectors/tests/Sandbox.TcoInspectors.Wpf/MainWindowViewModel.cs?name=DialogProxyServiceInitialization)]
    </example>
    </docu>
~*)
FUNCTION_BLOCK TcoDigitalInspector EXTENDS TcoInspector IMPLEMENTS ITcoDigitalInspector
VAR
    _data : TcoDigitalInspectorData;
END_VAR

(*~
    <docu>
        <summary>
            Gets common data settings of inspectors.
        </summary>
    </docu>
~*)
PROPERTY CommonData : REFERENCE TO TcoInspectorData
GET
CommonData REF= _data;
END_GET
END_PROPERTY

(*~
<docu>
<summary>
    Gets data of this inspector.
</summary>
</docu>
~*)
PROPERTY Data : REFERENCE TO TcoDigitalInspectorData
GET
Data REF= _data;
END_GET
END_PROPERTY

(*~
<docu>
<summary>
    Inspects the signal and evaluates that it matches the value set in `RequiredStatus`.
</summary>
<returns>
    Returns the interface with information about the state of inspection.
</returns>
</docu>
~*)
METHOD Inspect : IInspector
VAR_INPUT
    Status : BOOL;
END_VAR
Inspect := THIS^;
_inspectorTask.InspectionData REF= _data;
OnEnterInspection();

IF (IsOverinspected()) THEN
    RETURN;
END_IF

_inspectorTask.Invoke();

IF (_inspectorTask.Execute()) THEN
    IF (_data.IsByPassed) THEN
        _data.Result := eInspectorResult.Bypassed;
        _data.TimeStamp := Context.RealTimeClock.NowLocal();
        _inspectorTask.DoneWhen(TRUE);
        RETURN;
    END_IF

    _data.Result := eInspectorResult.Running;
    _inspectorTask._failTimer(IN := TRUE, PT := _data.FailTime);
    _inspectorTask._passTimer(IN := Status = _data.RequiredStatus, PT := _data.PassTime);
    _data.DetectedStatus := Status;

    IF (_inspectorTask._failTimer.Q OR _inspectorTask._passTimer.Q) THEN
        _inspectorTask.DoneWhen(TRUE);
        OnDone();
    END_IF;
END_IF;
END_METHOD

(*~
    <docu>
        <summary>
            Executes when task reaches the ```Done``` state .
        </summary>
    </docu>
~*)
METHOD PROTECTED OnDone
IF (_data.Result = eInspectorResult.Failed) THEN
    _data.DetectedStatus := NOT _data.RequiredStatus;
END_IF
END_METHOD

METHOD WithCoordinator : ITcoDigitalInspector
VAR_INPUT
    inCoordinator : TcoCore.ITcoCoordinator;
END_VAR
_WithCoordinator(inCoordinator);
WithCoordinator := THIS^;
END_METHOD

END_FUNCTION_BLOCK

// ---- POUs/TcoInspectionGroup/TcoInspectionGroup.TcPOU
FUNCTION_BLOCK TcoInspectionGroup EXTENDS TcoInspector IMPLEMENTS ITcoInspectionGroup, ITcoInspectionGroupAct
VAR
    {attribute 'hide'}
    _done                     : BOOL;				
    {attribute 'hide'}
    _done_PV                  : BOOL;				
    _overallResult            : TcoComprehensiveResult;
    _currentRunResult         : TcoComprehensiveResult;
    _inspections              : ARRAY[0..LAST_INSPECTION_INDEX] OF ULINT;
	_inspectionsEmpty         : ARRAY[0..LAST_INSPECTION_INDEX] OF ULINT;
    _inspectionIndex          : INT;
    _tierAct                  : TcoCore.TcoTier(THIS^);
    _normalizedAllowedRetries : UINT;
	
	
END_VAR

VAR CONSTANT
    LAST_INSPECTION_INDEX : INT := 50;
	MAX_NORMALIZED_RETRIES : UINT := 65535;
END_VAR

VAR 
	count : ULINT;
END_VAR

(*~
	<summary>
		Initiates grouped inspection.
	</summary>
~*)
METHOD Act : ITcoInspectionGroup
//VAR_IN_OUT
//	inoResult : TcoComprehensiveResult;
//END_VAR
OverInspected := FALSE;
_inspectionIndex          := 0;
_done                     := TRUE; // True then set to false if any inspector not done.
_normalizedAllowedRetries := MAX_NORMALIZED_RETRIES;
Act := THIS^;



IF (_tierAct.IsNewTier()) THEN
	_inspections:=_inspectionsEmpty;
    ClearResult(_currentRunResult);
END_IF
END_METHOD

METHOD ClearResult
VAR_IN_OUT
	inoResult : TcoComprehensiveResult;
END_VAR
inoResult.ErrorCodes := '';
inoResult.Failures := '';
inoResult.Result := eOverallResult.NoAction;
END_METHOD

(*~
	<docu>
		<summary>
			Gets common data settings of inspectors.
		</summary>			
	</docu>	
~*)
PROPERTY CommonData : REFERENCE TO TcoInspectorData
GET
VAR
	_data : TcoInspectorData; 
END_VAR
CommonData REF= _data;
END_GET
END_PROPERTY

METHOD Dialog : BOOL
VAR_INPUT
	inRetryStep : INT;
END_VAR
IF(THIS^.Done) THEN
	_tcoInspectorDialogue.OverInspected := THIS^.OverInspected;		
	IF(THIS^._currentRunResult.Result = eOverallResult.Failed) THEN
		THIS^._tcoInspectorDialogue.Invoke();
		_tcoInspectorDialogue();	
		
		{warning disable C0357}
		IF(_tcoInspectorDialogue._dialogRetry) THEN			
			Retry(inRetryStep);			
		END_IF
		
		IF(_tcoInspectorDialogue._dialogTerminate) THEN
			Terminate();
		END_IF
		
		IF(_tcoInspectorDialogue._dialogOverride) THEN
			CarryOn();
		END_IF
		{warning enable C0357}
	ELSE
		IF(Coordinator <> 0) THEN
			Coordinator.MoveNext();
		END_IF;	
	END_IF;	
END_IF;
END_METHOD

METHOD DialogWithExternalClose : BOOL
VAR_INPUT
	inRetryStep : INT;
	inRetrySignal:BOOL;
	inTerminateSignal : BOOL;
END_VAR
//IF THIS^._tcoInspectorDialogue.State=eTaskState.Ready THEN
//	THIS^._tcoInspectorDialogue.DialogRetry 	    :=  FALSE;	
//	THIS^._tcoInspectorDialogue.DialogTerminate  	:=  FALSE;	
//	THIS^._tcoInspectorDialogue.DialogOverride   	:=  FALSE;
//END_IF




_tcoInspectorDialogue.HandleExternalSignals(inRetrySignal:=inRetrySignal,inTerminateSignal:=inTerminateSignal);


IF(THIS^.Done) THEN
	_tcoInspectorDialogue.OverInspected := THIS^.OverInspected;		
	IF(THIS^._currentRunResult.Result = eOverallResult.Failed) THEN
		THIS^._tcoInspectorDialogue.Invoke();
		_tcoInspectorDialogue();	
						
		
		{warning disable C0357}
		IF(_tcoInspectorDialogue._dialogRetry AND _tcoInspectorDialogue.DialogIsClosed ) THEN			
			Retry(inRetryStep);	
	
		END_IF
		
		IF(_tcoInspectorDialogue._dialogTerminate AND _tcoInspectorDialogue.DialogIsClosed ) THEN
			Terminate();
		END_IF
		
		IF(_tcoInspectorDialogue._dialogOverride AND _tcoInspectorDialogue.DialogIsClosed) THEN
			CarryOn();
		END_IF
		{warning enable C0357}
	ELSE
		IF(Coordinator <> 0) THEN
			Coordinator.MoveNext();
		END_IF;	
	END_IF;	
END_IF;

IF THIS^._tcoInspectorDialogue.State=eTaskState.Done 
		AND ( _tcoInspectorDialogue.DialogRetry
		OR _tcoInspectorDialogue.DialogTerminate
		OR _tcoInspectorDialogue.DialogOverride)
		AND _tcoInspectorDialogue.DialogIsClosed  THEN	
	THIS^._tcoInspectorDialogue.Restore();
END_IF;
END_METHOD

PROPERTY Done : BOOL
GET
Done := _done;
END_GET
END_PROPERTY

(*~
	<docu>
		<summary>
			Upon failure the inspection retries given number of time. When it reach	given numbers then terminate 		
		</summary>			
	</docu>	
~*)

{attribute 'hide'}
{attribute 'obsolete' := 'You should access `Evaluate` method via `OnFail()` method.'}
METHOD PUBLIC Evaluate : BOOL
VAR_INPUT
    (*~
	<docu>
		<summary>
			State from which the inspection will restart.		
		</summary>			
	</docu>	
	~*)
    inFromState : INT;
    (*~
	<docu>
		<summary>
			Behavior when ispection is failed		
		</summary>			
	</docu>	
	~*)
    inFailMode : eTcoInspectorFailMode;
    (*~
	<docu>
		<summary>
			State from which the inspection will continue.		
		</summary>			
	</docu>	
	~*)
    inToState : INT;
END_VAR
IF (_coordinator = 0) THEN
    RETURN;
END_IF

IF (THIS^.Done) THEN
    IF (THIS^._currentRunResult.Result = eOverallResult.Failed) THEN
        IF (__ISVALIDREF(_refOverallResult)) THEN
            _refOverallResult := _originalOverallResult;
        END_IF

        IF inFailMode = eTcoInspectorFailMode.CarryOn THEN
            _coordinator.MoveNext();
        ELSIF inFailMode = eTcoInspectorFailMode.JumpTo THEN
            _coordinator.Retry(inToState);
        ELSIF inFailMode = eTcoInspectorFailMode.Terminate THEN
            _coordinator.Terminate();
        ELSIF inFailMode = eTcoInspectorFailMode.RetryThenCarryOn THEN
            IF OverInspected THEN
                _coordinator.MoveNext();
            ELSE
                _coordinator.Retry(inFromState);
            END_IF;
        ELSIF inFailMode = eTcoInspectorFailMode.RetryThenJumpTo THEN
            IF OverInspected THEN
                _coordinator.Retry(inToState);
            ELSE
                _coordinator.Retry(inFromState);
            END_IF;

        ELSIF inFailMode = eTcoInspectorFailMode.RetryThenTeminate THEN
            IF OverInspected THEN
                _coordinator.Terminate();
            ELSE
                _coordinator.Retry(inFromState);
            END_IF;

        END_IF
    ELSE

        _coordinator.MoveNext();
    END_IF;
END_IF;

Evaluate := THIS^.Done;
END_METHOD

(*~
	<summary>
		Add inspector to inspection group to inspect
	</summary>
~*)
METHOD Inspect : ITcoInspectionGroup
VAR_INPUT
    Inspector : IInspector;
END_VAR
OnEnterInspection();

IF(_normalizedAllowedRetries <> 0 
AND _normalizedAllowedRetries <> MAX_NORMALIZED_RETRIES) THEN
	Inspector.CommonData.NumberOfAllowedRetries := _normalizedAllowedRetries;
END_IF;

Inspect := THIS^;


IF(Inspector.OverInspected) THEN
	THIS^.OverInspected := TRUE;
END_IF;

IF (Inspector.Done) THEN
    Inspector.UpdateComprehensiveResult(_currentRunResult);							
ELSE
	_done := FALSE;	
	_done_PV := FALSE;	
END_IF


IF(_inspectionIndex < LAST_INSPECTION_INDEX)THEN
	_inspections[_inspectionIndex] :=  Inspector.Identity;
	_inspectionIndex := _inspectionIndex + 1;
END_IF
END_METHOD

(*~
	<summary>
		Sets lower `number of allowed retries` for this call of inspection group.
		Invoke this method multiple times if you want to check for the inspection for lowest numebr of retries.
		<note type="important">
			The inspections will run at least once before allowed entries is normalized.
		</note>
	</summary>
~*)

METHOD NormalizeRetries : ITcoInspectionGroup
VAR_INPUT
	inoInspection : IInspector;
END_VAR
// Determine lowest number of retries
NormalizeRetries := THIS^;
IF( inoInspection.CommonData.NumberOfAllowedRetries <> 0 
AND_THEN inoInspection.CommonData.NumberOfAllowedRetries < _normalizedAllowedRetries) THEN
	_normalizedAllowedRetries := inoInspection.CommonData.NumberOfAllowedRetries;
END_IF
END_METHOD

METHOD OnFail : IOnFail
VAR_INPUT
END_VAR
//THIS^._tcoInspectorDialogue.SetInspector(THIS^);
OnFail := THIS^;
END_METHOD

(*~
	<docu>
		<summary>
			Gets `true` when the number of inspections excceds `NumberOfAllowedRetries`.
		</summary>			
	</docu>	
~*)
PROPERTY PUBLIC OverInspected : BOOL
GET
OverInspected := _isOverInspected;
END_GET
SET
_isOverInspected := OverInspected;
END_SET
END_PROPERTY

{attribute 'hide'}
{attribute 'obsolete' := 'You should access `Retry` method via `OnFail()` method.'}
METHOD Retry : BOOL
VAR_INPUT
	inFromState : INT;
END_VAR
IF(_coordinator = 0) THEN
	RETURN;	
END_IF

IF(THIS^.Done) THEN
	IF(THIS^._currentRunResult.Result = eOverallResult.Failed) THEN		
		IF(__ISVALIDREF(_refOverallResult)) THEN
			_refOverallResult := _originalOverallResult;
		END_IF	 
		ClearResult(_currentRunResult);	   	
		_coordinator.Retry(inFromState);
	ELSE
		_coordinator.MoveNext();
	END_IF;	
END_IF;	


Retry := THIS^.Done;
END_METHOD

{attribute 'hide'}
{attribute 'obsolete' := 'You should access `RetryThenTerminate` method via `OnFail()` method.'}
METHOD RetryThenTerminate : BOOL
VAR_INPUT
	inFromState : INT;
END_VAR
IF (_coordinator = 0) THEN
    RETURN;
END_IF

IF (THIS^.Done) THEN
    IF (THIS^._currentRunResult.Result = eOverallResult.Failed) THEN
        IF (__ISVALIDREF(_refOverallResult)) THEN
            _refOverallResult := _originalOverallResult;
        END_IF

        ClearResult(_currentRunResult);
        IF OverInspected THEN
            _coordinator.Terminate();
        ELSE
            _coordinator.Retry(inFromState);
        END_IF;
    ELSE
        _coordinator.MoveNext();
    END_IF;
END_IF;

RetryThenTerminate := THIS^.Done;
END_METHOD

{attribute 'hide'}
{attribute 'obsolete' := 'You should access `Terminate` method via `OnFail()` method.'}
METHOD Terminate : BOOL
IF(_coordinator = 0) THEN
	RETURN;	
END_IF

IF(THIS^.Done) THEN
	IF(THIS^._currentRunResult.Result = eOverallResult.Failed) THEN
		_coordinator.Terminate();
	ELSE
		_coordinator.MoveNext();
	END_IF;	
END_IF;	

Terminate := THIS^.Done;
END_METHOD

(*~
	<docu>
		<summary>
			Updates comprehensive result. The comprehensive result is set to `Failed` when any inspection fails or is inconclusive.
			Any bypassed or excluded inspection are not taken in the account.			
		</summary>			
	</docu>	
~*)

METHOD UpdateComprehensiveResult : IInspector
VAR_IN_OUT
	(*~
	<docu>
		<summary>
			Comprehensive result data structure to be updated.	
		</summary>			
	</docu>	
	~*)
    inoResult : TcoComprehensiveResult;
END_VAR
UpdateComprehensiveResult := THIS^;

_refOverallResult REF= inoResult;

IF(_tierUpdateOverall.IsNewTier()) THEN	
	_originalOverallResult := inoResult;
END_IF

		
CASE _currentRunResult.Result OF
	eOverallResult.NoAction:
		;
	eOverallResult.Passed:
		;
	eOverallResult.Failed:
		 
		_refOverallResult.Result		:= eOverallResult.Failed;
		_refOverallResult.Failures		:= _currentRunResult.Failures;
		_refOverallResult.ErrorCodes	:= _currentRunResult.ErrorCodes;
END_CASE


IF(_done) THEN
	_overallResult := _refOverallResult;
END_IF;
END_METHOD

(*~
	<docu>
		<summary>
			Updates failure description. Adding `FailureDescription` do the overall result structure.
		</summary>	
	</docu>	
~*)
METHOD PROTECTED UpdateDescriptions
VAR_IN_OUT
	inoResult : TcoComprehensiveResult;
END_VAR
IF NOT _done THEN
	_done_PV := FALSE;	
END_IF
IF(_done AND NOT _done_PV) THEN
	inoResult.Failures := THIS^.Context.Environment.Messaging.StringBuilder.Clear()
				.Append(inoResult.Failures)				
				.Append(CommonData.FailureDescription)
				.Append(';')
				.ToString();
	
	inoResult.ErrorCodes := THIS^.Context.Environment.Messaging.StringBuilder.Clear()
				.Append(inoResult.ErrorCodes)				
				.Append(CommonData.ErrorCode)
				.Append(';')
				.ToString();			
	_done_PV := TRUE;	
END_IF;
END_METHOD

METHOD WithCoordinator : ITcoInspectionGroupAct
VAR_INPUT
	inCoordinator : TcoCore.ITcoCoordinator;
END_VAR
_WithCoordinator(inCoordinator);
WithCoordinator := THIS^;
END_METHOD

END_FUNCTION_BLOCK
